TYPE DUT_MotionStage :
    // Defines the EPICS interface to moving a motor in TwinCAT
STRUCT
    (* Hardware *)

    // PLC Axis Reference
    Axis: AXIS_REF;
    // NC Forward Limit Switch: TRUE if ok to move
    {attribute 'pytmc' := '
        pv: PLC:bLimitForwardEnable
        io: i
        field: ZNAM FALSE
        field: ONAM TRUE
        field: DESC FALSE if forward limit hit
    '}
    bLimitForwardEnable AT %I*: BOOL;
    // NC Backward Limit Switch: TRUE if ok to move
    {attribute 'pytmc' := '
        pv: PLC:bLimitBackwardEnable
        io: i
        field: ZNAM FALSE
        field: ONAM TRUE
        field: DESC FALSE if reverse limit hit
    '}
    bLimitBackwardEnable AT %I*: BOOL;
    // NO Home Switch: TRUE if at home
    {attribute 'pytmc' := '
        pv: PLC:bHome
        io: i
        field: ZNAM FALSE
        field: ONAM TRUE
        field: DESC TRUE if at homing switch
    '}
    bHome AT %I*: BOOL;
    // NC Brake Output: TRUE to release brake
    {attribute 'pytmc' := '
        pv: PLC:bBrakeRelease
        io: i
        field: ZNAM FALSE
        field: ONAM TRUE
        field: DESC TRUE if brake released
    '}
    bBrakeRelease AT %Q*: BOOL;
    // NC STO Input: TRUE if ok to move
    {attribute 'pytmc' := '
        pv: PLC:bHardwareEnable
        io: i
        field: ZNAM FALSE
        field: ONAM TRUE
        field: DESC TRUE if STO not hit
    '}
    bHardwareEnable AT %I*: BOOL;

    // Raw encoder IO for ULINT (Biss-C)
    nRawEncoderULINT AT %I*: ULINT;
    // Raw encoder IO for UINT (Relative Encoders)
    nRawEncoderUINT AT %I*: UINT;
    // Raw encoder IO for INT (LVDT)
    nRawEncoderINT AT %I*: INT;

    (* Psuedo-hardware *)

    // Forward enable EPS summary
    {attribute 'pytmc' := '
        pv: PLC:bAllForwardEnable
        io: i
        field: ZNAM FALSE
        field: ONAM TRUE
        field: DESC Summary of axis permission to move forward
    '}
    bAllForwardEnable: BOOL:=FALSE;
    // Backward enable EPS summary
    {attribute 'pytmc' := '
        pv: PLC:bAllBackwardEnable
        io: i
        field: ZNAM FALSE
        field: ONAM TRUE
        field: DESC Summary of axis permission to move backward
    '}
    bAllBackwardEnable: BOOL:=FALSE;
    // Enable EPS summary encapsulating emergency stop button and any additional motion preventive hardware
    {attribute 'pytmc' := '
        pv: PLC:bAllEnable
        io: i
        field: ZNAM FALSE
        field: ONAM TRUE
        field: DESC Summary of axis permission to have power
    '}
    bAllEnable: BOOL:=FALSE;
    // Forward virtual gantry limit switch
    {attribute 'pytmc' := '
        pv: PLC:bGantryForwardEnable
        io: i
        field: ZNAM FALSE
        field: ONAM TRUE
        field: DESC TRUE if gantry ok to move forward
    '}
    bGantryForwardEnable: BOOL:=FALSE;
    // Backward virtual gantry limit switch
    {attribute 'pytmc' := '
        pv: PLC:bGantryBackwardEnable
        io: i
        field: ZNAM FALSE
        field: ONAM TRUE
        field: DESC TRUE if gantry ok to move backward
    '}
    bGantryBackwardEnable: BOOL:=FALSE;
    // Encoder count summary, if linked above
    {attribute 'pytmc' := '
        pv: PLC:nEncoderCount
        io: i
        field: DESC Count from encoder hardware
    '}
    nEncoderCount: UDINT;
	
	// Forward Enable EPS struct
	{attribute 'pytmc' := '
        pv: PLC:stEPSForwardEnable
        io: i
        field: DESC Forward Enable Interlocks
    '}
	stEPSForwardEnable: DUT_EPS;
	
	// Backward Enable EPS struct
	{attribute 'pytmc' := '
        pv: PLC:stEPSBackwardEnable
        io: i
        field: DESC Backward Enable Interlocks
    '}
	stEPSBackwardEnable: DUT_EPS;
	
	// Power Enable EPS struct
	{attribute 'pytmc' := '
        pv: PLC:stEPSPowerEnable
        io: i
        field: DESC Power Interlocks
    '}
	stEPSPowerEnable: DUT_EPS;

    (* Settings *)
    // Name to use for log messages, fast faults, etc.
    {attribute 'pytmc' := '
        pv: PLC:sName
        io: i
        field: DESC PLC program name
    '}
    sName: STRING;
    // If TRUE, we want to enable the motor independently of PMPS or other safety systems.
    {attribute 'pytmc' := '
        pv: PLC:bPowerSelf
        io: i
        field: ZNAM FALSE
        field: ONAM TRUE
        field: DESC FALSE if axis is in PMPS
    '}
    bPowerSelf: BOOL:=FALSE;
    // Determines when we automatically enable the motor
    {attribute 'pytmc' := '
        pv: PLC:nEnableMode
        io: i
        field: DESC Describes when the axis will automatically get power
    '}
    nEnableMode: ENUM_StageEnableMode:=ENUM_StageEnableMode.DURING_MOTION;
    // Determines when we automatically disengage the brake
    {attribute 'pytmc' := '
        pv: PLC:nBrakeMode
        io: i
        field: DESC Describes when the brake will be released
    '}
    nBrakeMode: ENUM_StageBrakeMode:=ENUM_StageBrakeMode.IF_ENABLED;
    // Determines our encoder homing strategy
    {attribute 'pytmc' := '
        pv: PLC:nHomingMode
        io: i
        field: DESC Describes our homing strategy
    '}
    nHomingMode: ENUM_EpicsHomeCmd:=ENUM_EpicsHomeCmd.NONE;
    // Set true to activate gantry EPS
    {attribute 'pytmc' := '
        pv: PLC:bGantryAxis
        io: i
        field: ZNAM FALSE
        field: ONAM TRUE
        field: DESC TRUE if gantry EPS active
    '}
    bGantryAxis: BOOL:=FALSE;

    // Set to gantry difference tolerance
    nGantryTol: LINT:=0;

    // Encoder count at which this axis is aligned with other axis
    nEncRef: ULINT:=0;

    (* Commands *)
    // Used internally to request enables
    {attribute 'pytmc' := '
        pv: PLC:bEnable
        io: io
        field: ZNAM FALSE
        field: ONAM TRUE
        field: DESC Used internally to request enables
    '}
    bEnable: BOOL;
    // Used internally to reset errors and other state
    {attribute 'pytmc' := '
        pv: PLC:bReset
        io: io
        field: ZNAM FALSE
        field: ONAM TRUE
        field: DESC Used internally to reset errors
    '}
    bReset: BOOL;
    // Used internally and by the IOC to start or stop a move
    {attribute 'pytmc' := '
        pv: PLC:bExecute
        io: io
        field: ZNAM FALSE
        field: ONAM TRUE
        field: DESC Used internally and by the IOC to start or stop
    '}
    bExecute: BOOL;
    // Used by the IOC to disable an axis
    {attribute 'pytmc' := '
        pv: PLC:bUserEnable
        io: io
        field: ZNAM DISABLE
        field: ONAM ENABLE
        field: DESC Used to disable power entirely for an axis
    '}
    bUserEnable: BOOL := 1;

    (* Shortcut Commands *)
    // Start a move to fPosition with fVelocity
    {attribute 'pytmc' := '
        pv: PLC:bMoveCmd
        io: io
        field: DESC Start a move
    '}
    bMoveCmd: BOOL;
    // Start the homing routine
    {attribute 'pytmc' := '
        pv: PLC:bHomeCmd
        io: io
        field: DESC Start the homing routine
    '}
    bHomeCmd: BOOL;

    (* Command Args *)
    // Used internally and by the IOC to pick what kind of move to do
    {attribute 'pytmc' := '
        pv: PLC:nCommand
        io: io
        field: DESC Used internally and by the IOC to pick move type
    '}
    nCommand: INT;
    // Used internally and by the IOC to pass additional data to some commands
    {attribute 'pytmc' := '
        pv: PLC:nCmdData
        io: io
        field: DESC Used internally and by the IOC to pass extra args
    '}
    nCmdData: INT;
    // Used internally and by the IOC to pick a destination for the move
    {attribute 'pytmc' := '
        pv: PLC:fPosition
        io: io
        field: DESC Used internally and by the IOC as the set position
    '}
    fPosition: LREAL;
    // Used internally and by the IOC to pick a move velocity
    {attribute 'pytmc' := '
        pv: PLC:fVelocity
        io: io
        field: DESC Used internally and by the IOC to set velocity
    '}
    fVelocity: LREAL;
    // Used internally and by the IOC to pick a move acceleration
    {attribute 'pytmc' := '
        pv: PLC:fAcceleration
        io: io
        field: DESC Used internally and by the IOC to set acceleration
    '}
    fAcceleration: LREAL;
    // Used internally and by the IOC to pick a move deceleration
    {attribute 'pytmc' := '
        pv: PLC:fDeceleration
        io: io
        field: DESC Used internally and by the IOC to set deceleration
    '}
    fDeceleration: LREAL;
    // Used internally and by the IOC to pick a home position
    {attribute 'pytmc' := '
        pv: PLC:fHomePosition
        io: io
        field: DESC Used internally and by the IOC to pick home position
    '}
    fHomePosition: LREAL;

    (* Info *)
    // Unique ID assigned to each axis in the NC
    {attribute 'pytmc' := '
        pv: PLC:nMotionAxisID
        io: i
        field: DESC Unique ID assigned to each axis in the NC
    '}
    nMotionAxisID: UDINT:=0;

    (* Returns *)
    // TRUE if done enabling
    {attribute 'pytmc' := '
        pv: PLC:bEnableDone
        io: i
        field: ZNAM FALSE
        field: ONAM TRUE
        field: DESC TRUE if done enabling
    '}
    bEnableDone: BOOL;
    // TRUE if in the middle of a command
    {attribute 'pytmc' := '
        pv: PLC:bBusy
        io: i
        field: ZNAM FALSE
        field: ONAM TRUE
        field: DESC TRUE if in the middle of a command
    '}
    bBusy: BOOL;
    // TRUE if we've done a command and it has finished
    {attribute 'pytmc' := '
        pv: PLC:bDone
        io: i
        field: ZNAM FALSE
        field: ONAM TRUE
        field: DESC TRUE if command finished successfully
    '}
    bDone: BOOL;
    // TRUE if the motor has been homed, or does not need to be homed
    {attribute 'pytmc' := '
        pv: PLC:bHomed
        io: i
        field: DESC TRUE if the motor has been homed
    '}
    bHomed: BOOL;
    // TRUE if we have safety permission to move
    {attribute 'pytmc' := '
        pv: PLC:bSafetyReady
        io: i
        field: ZNAM FALSE
        field: ONAM TRUE
        field: DESC TRUE if safe to start a move
    '}
    bSafetyReady: BOOL;
    // TRUE if we're in an error state
    {attribute 'pytmc' := '
        pv: PLC:bError
        io: i
        field: ZNAM FALSE
        field: ONAM TRUE
        field: DESC TRUE if we are in an error state
        update: 100Hz notify
    '}
    bError: BOOL;
    // Error code if nonzero
    {attribute 'pytmc' := '
        pv: PLC:nErrorId
        io: i
        field: DESC Error code if nonzero
        update: 100Hz notify
    '}
    nErrorId: UDINT;
    // Message to identify the error state
    {attribute 'pytmc' := '
        pv: PLC:sErrorMessage
        io: i
        field: DESC Message to identify the error state
        update: 100Hz notify
    '}
    sErrorMessage: STRING;
    // Internal hook for custom error messages
    sCustomErrorMessage: STRING;
    // MC_ReadParameterSet Output
    stAxisParameters: ST_AxisParameterSet;
    // True if we've updated stAxisParameters at least once
    bAxisParamsInit: BOOL;

    // Misc axis status information for the IOC
    stAxisStatus: DUT_AxisStatus_v0_01;

    (* Other status information for users of the IOC *)
    // Position lag difference
    {attribute 'pytmc' := '
        pv: PLC:fPosDiff
        io: i
        field: DESC Position lag difference
    '}
    fPosDiff: LREAL;
END_STRUCT
END_TYPE

(* stored: Version 1.1.0.1, ProductVersion 3.1.4024.12
   DUT DUT_MotionStage: Id {10b5775d-5646-4d55-ad77-40abc3888de3} *)
